(* IEC 61131-3 sources: RL_MAR/experiments/comparison/autoplc/results/deepseek-ai-DeepSeek-V3.2_20260508_111905/med_27, 1 file *)

(* ---- med_27_1.st ---- *)
FUNCTION_BLOCK FlowerArrangingMachine
VAR_INPUT
    FlowerTypeSensor : INT; (* Input for detecting flower type *)
    FlowerColorSensor : INT; (* Input for detecting flower color *)
END_VAR
VAR_OUTPUT
    ArrangingMechanism : INT; (* Output for controlling arranging mechanism *)
    ConveyorBelt : BOOL; (* Output for controlling conveyor belt *)
END_VAR

VAR
    // No internal variables needed for this simple combinatorial logic
END_VAR

// Main control logic
IF (FlowerTypeSensor = 1) AND (FlowerColorSensor = 1) THEN
    ArrangingMechanism := 1;  // red type 1 flower
ELSIF (FlowerTypeSensor = 1) AND (FlowerColorSensor = 2) THEN
    ArrangingMechanism := 2;  // blue type 1 flower
ELSIF (FlowerTypeSensor = 2) AND (FlowerColorSensor = 1) THEN
    ArrangingMechanism := 3;  // red type 2 flower
ELSIF (FlowerTypeSensor = 2) AND (FlowerColorSensor = 2) THEN
    ArrangingMechanism := 4;  // blue type 2 flower
ELSE
    ArrangingMechanism := 0;  // any other combination
END_IF

// Conveyor belt control based on arranging mechanism
IF ArrangingMechanism <> 0 THEN
    ConveyorBelt := TRUE;
ELSE
    ConveyorBelt := FALSE;
END_IF

END_FUNCTION_BLOCK
